FUNCTION_BLOCK fbTest IMPLEMENTS I_Observable

END_FUNCTION_BLOCK

(* stored: Version 1.1.0.1, ProductVersion 3.1.4024.11
   POU fbTest: Id {507e757d-b58f-4376-a86c-3c62448a9975}, SpecialFunc None *)
